FUNCTION_BLOCK FB_Bel
VAR_INPUT
	Freigabe_auto			: BOOL;
	Freigabe_Deakt_auto		: BOOL;
	Betrieb_Anford_auto		: BOOL;
	Steuerung_Sollw_auto	: REAL; (* 0-100*)
	Quittierung				: BOOL;
	Adresse					: BYTE;
	AdressType				: E_DALIV2AddrType;
END_VAR
VAR_OUTPUT
	Steuerung				: ST_Bel_Steuerung;
	Stellwert				: ST_Bel_Stellwert;
	Zustand					: ST_Bel_Zustand;
	Parameter				: ST_Bel_Parameter;
END_VAR
VAR
	Zustandscheck			: FB_Bel_Zustandscheck;
	Logik					: FB_Bel_Logik;
	Ablaufsteuerung			: FB_Bel_Ablaufsteuerung;
	Sollwertscheck			: FB_Bel_Sollwertscheck;
	SteuerungsVorgang		: FB_Bel_Steuerung;

	Stellwertscheck			: FB_Bel_Stellwertscheck;
	QuitTrig				: FB_SetResetFallTrigger;

	LeseDaten				: FB_Bel_Input;
	SchreibeDaten			: FB_Bel_Output;

	Dali_Dimmer				: FB_DALIV2Dimmer1Switch;
	Dali_Communication		: FB_DALIV2Communication;
	Dali_Off				: FB_DALIV2Off;
	Dali_ArcPower			: FB_DALIV2DirectArcPowerControl;

	OUT_Dali_Betrieb		: BOOL;
	OUT_Dali_Leistung		: BYTE;
	Dali_Error				: BOOL;
	Dali_Dimm_Betrieb		: BOOL:= FALSE;
	Dali_ErrorID			: UDINT;
	Dali_bBusy				: BOOL;
	Dali_bOn				: BOOL:=TRUE;
	Dali_bOff				: BOOL:=FALSE;
	Dali_TON				: TON;

	Dali_Arc_Busy			: BOOL;
	Dali_Arc_Error			: BOOL;
	Dali_Arc_ErrorID		: UDINT;

	Dali_Off_Busy			: BOOL;
	Dali_Off_Error			: BOOL;
	Dali_Off_ErrorID		: UDINT;

	IN_Leistung				: BYTE;
	IN_Dali_Arc_Error		: BOOL;
	IN_Dali_Off_Error		: BOOL;
	IN_Dali_Error			: BOOL;

	DALI_GetSettings		: FB_DALIV2GetSettings;
	DALI_Setting_Array		: ARRAY [0..63] OF ST_DALIV2DeviceSettings;
	Lampen_Monitoring		: FB_Bel_Monitoring;

END_VAR

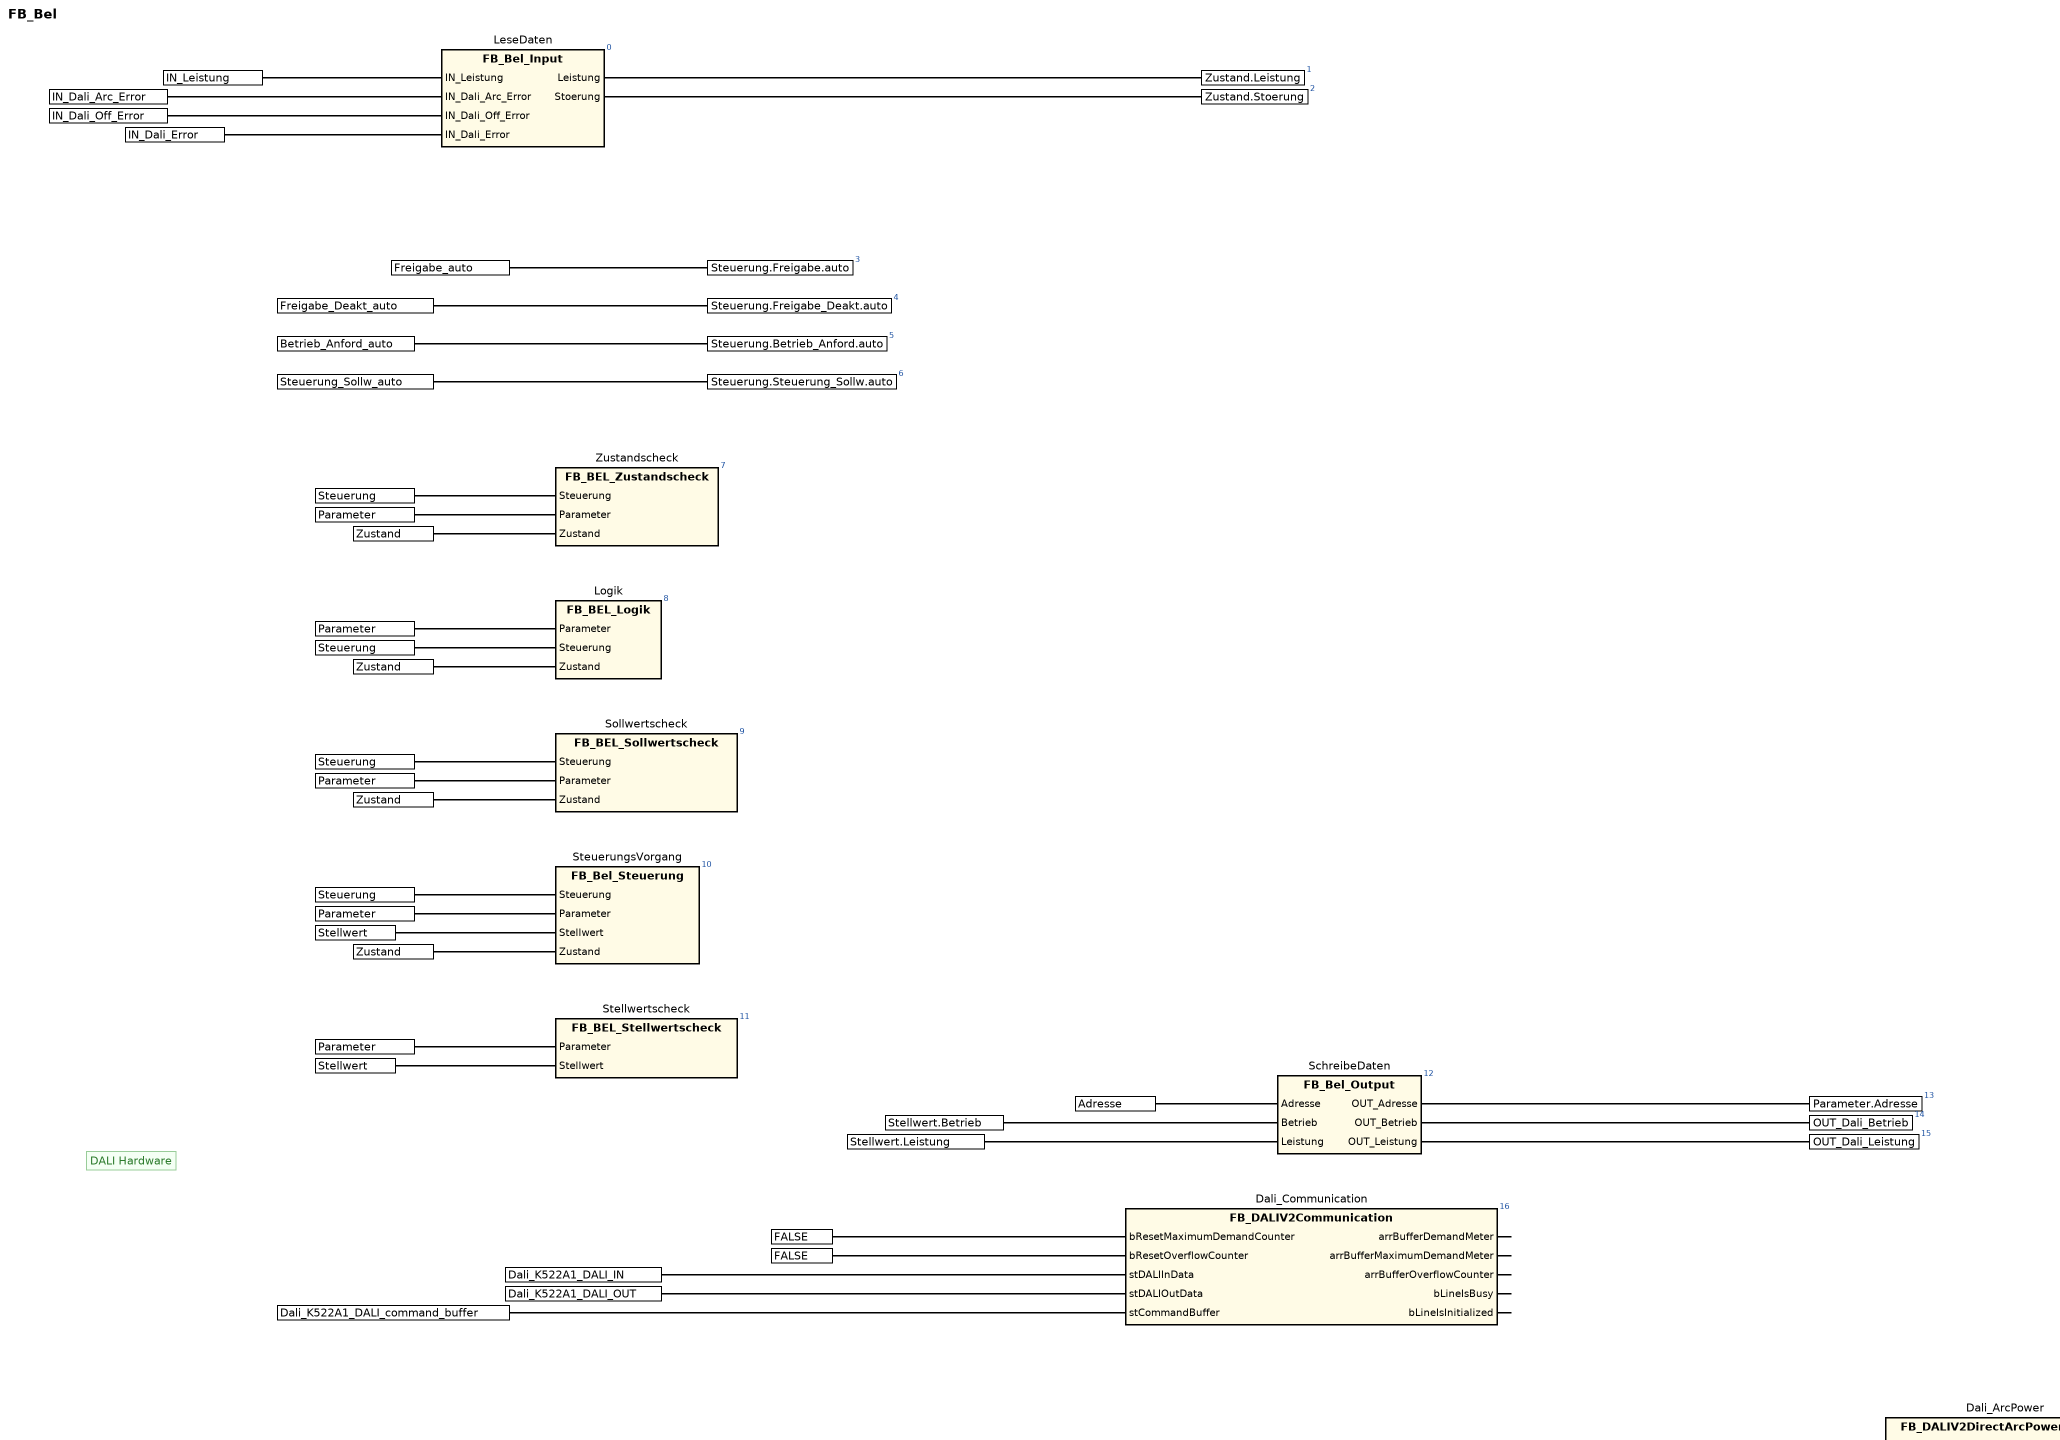
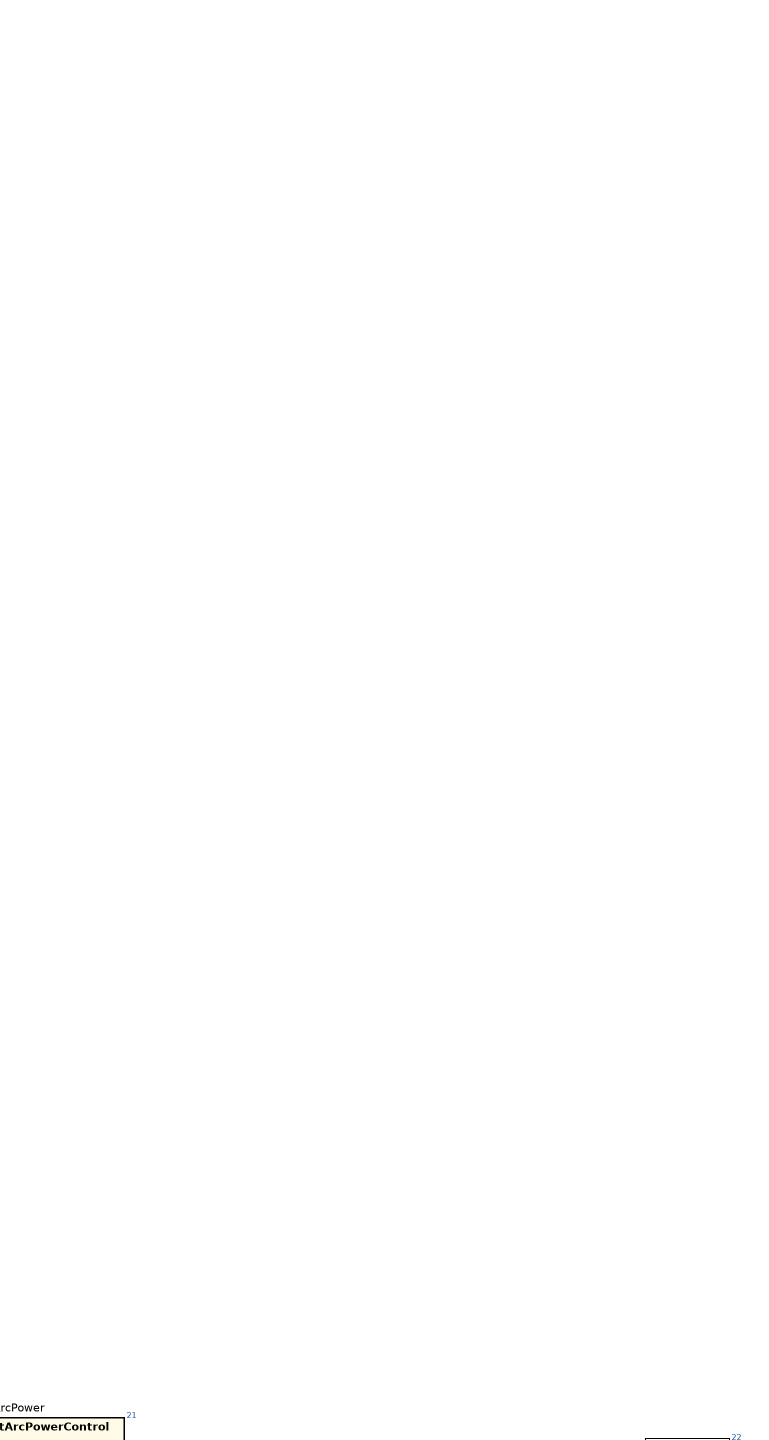
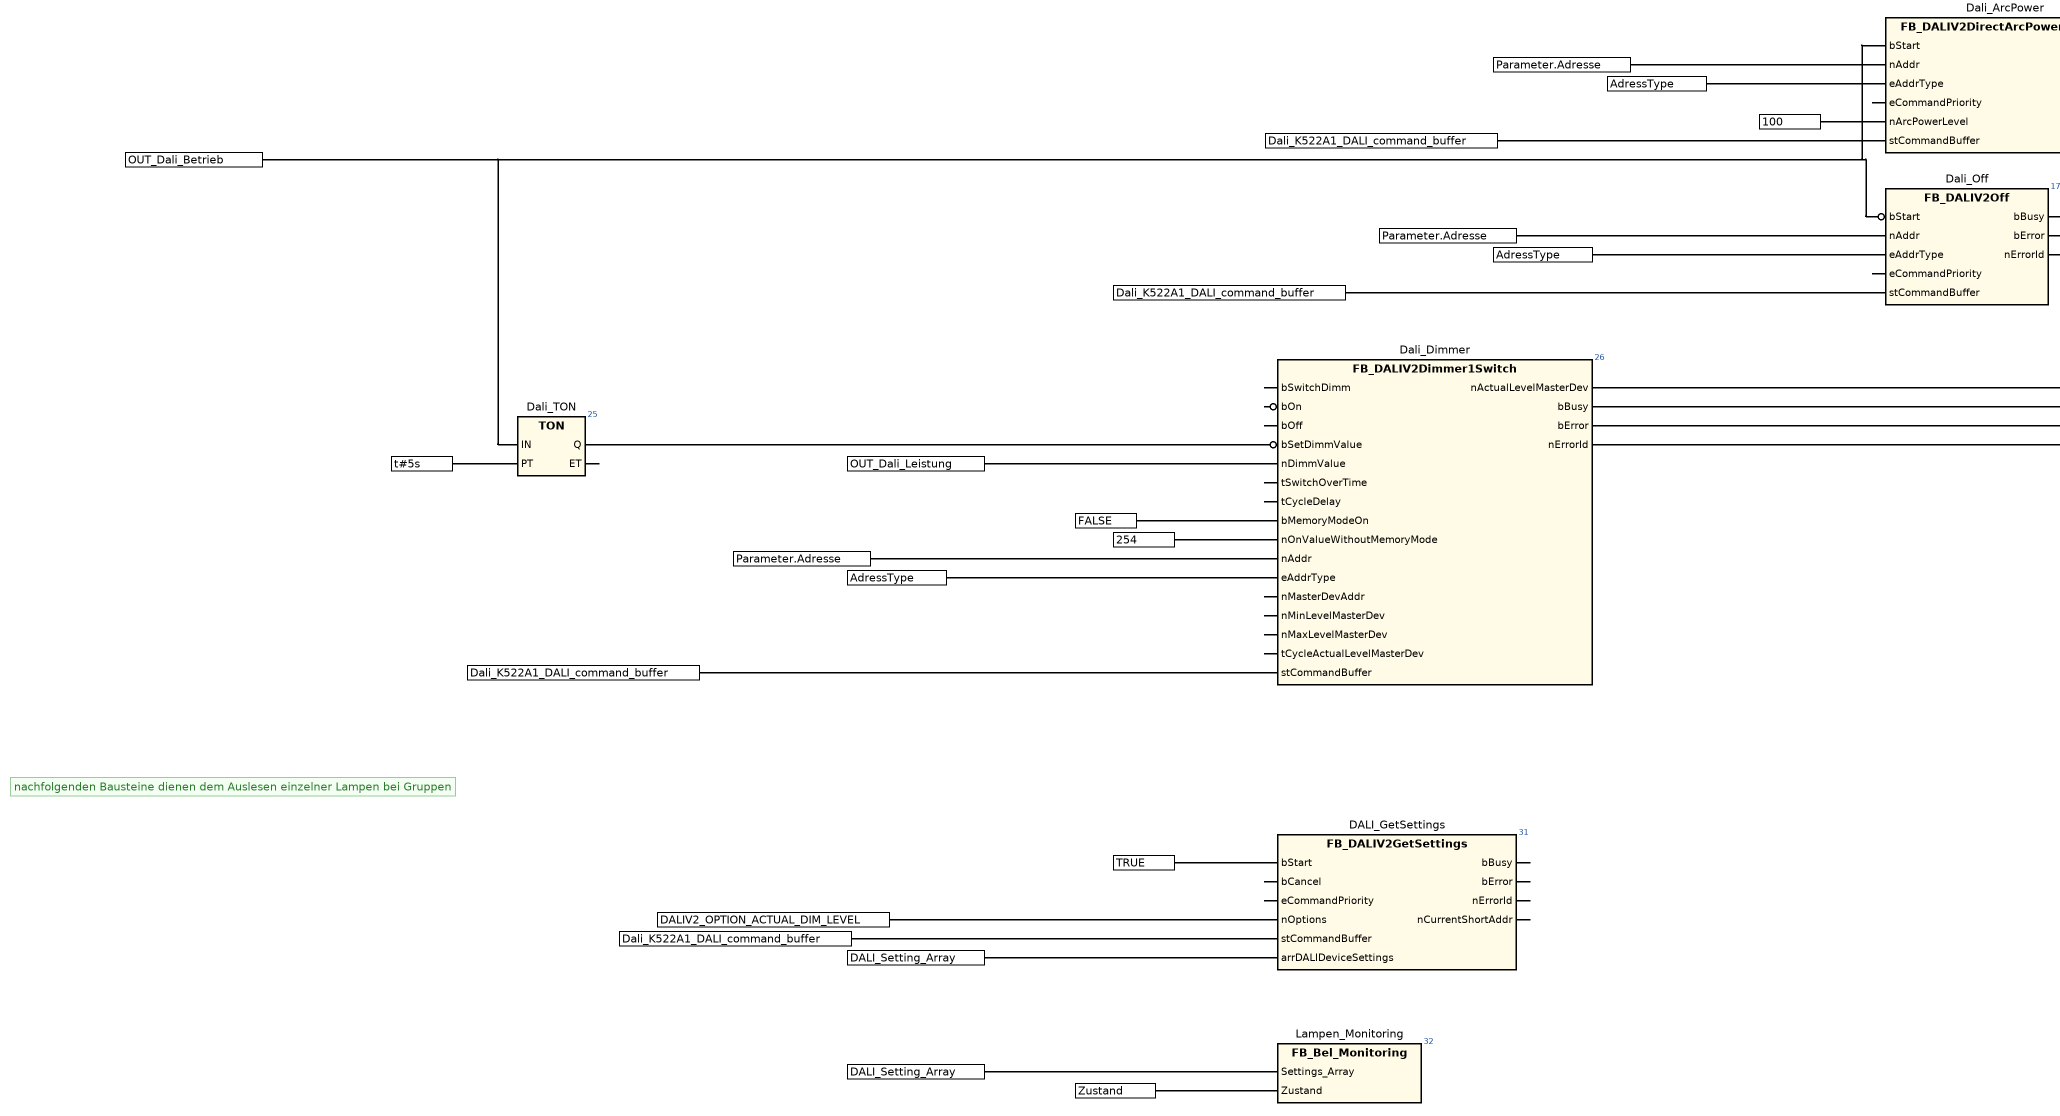
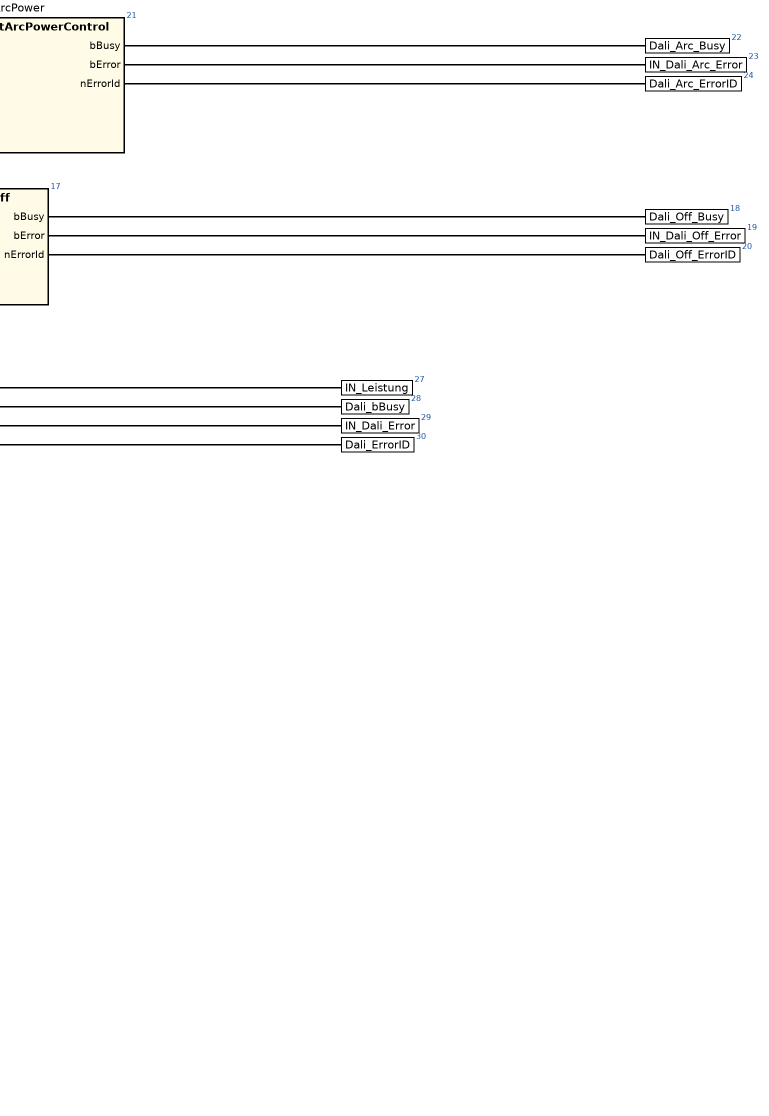
LeseDaten(
    IN_Leistung := IN_Leistung,
    IN_Dali_Arc_Error := IN_Dali_Arc_Error,
    IN_Dali_Off_Error := IN_Dali_Off_Error,
    IN_Dali_Error := IN_Dali_Error); // FB_Bel_Input
Zustand.Leistung := LeseDaten.Leistung;
Zustand.Stoerung := LeseDaten.Stoerung;
Steuerung.Freigabe.auto := Freigabe_auto;
Steuerung.Freigabe_Deakt.auto := Freigabe_Deakt_auto;
Steuerung.Betrieb_Anford.auto := Betrieb_Anford_auto;
Steuerung.Steuerung_Sollw.auto := Steuerung_Sollw_auto;
Zustandscheck(Steuerung := Steuerung, Parameter := Parameter, Zustand := Zustand); // FB_BEL_Zustandscheck
Logik(Parameter := Parameter, Steuerung := Steuerung, Zustand := Zustand); // FB_BEL_Logik
Sollwertscheck(Steuerung := Steuerung, Parameter := Parameter, Zustand := Zustand); // FB_BEL_Sollwertscheck
SteuerungsVorgang(Steuerung := Steuerung, Parameter := Parameter, Stellwert := Stellwert, Zustand := Zustand); // FB_Bel_Steuerung
Stellwertscheck(Parameter := Parameter, Stellwert := Stellwert); // FB_BEL_Stellwertscheck
SchreibeDaten(Adresse := Adresse, Betrieb := Stellwert.Betrieb, Leistung := Stellwert.Leistung); // FB_Bel_Output
Parameter.Adresse := SchreibeDaten.OUT_Adresse;
OUT_Dali_Betrieb := SchreibeDaten.OUT_Betrieb;
OUT_Dali_Leistung := SchreibeDaten.OUT_Leistung;
// DALI Hardware
Dali_Communication(
    bResetMaximumDemandCounter := FALSE,
    bResetOverflowCounter := FALSE,
    stDALIInData := Dali_K522A1_DALI_IN,
    stDALIOutData := Dali_K522A1_DALI_OUT,
    stCommandBuffer := Dali_K522A1_DALI_command_buffer); // FB_DALIV2Communication
Dali_Off(
    bStart := NOT OUT_Dali_Betrieb,
    nAddr := Parameter.Adresse,
    eAddrType := AdressType,
    stCommandBuffer := Dali_K522A1_DALI_command_buffer); // FB_DALIV2Off
Dali_Off_Busy := Dali_Off.bBusy;
IN_Dali_Off_Error := Dali_Off.bError;
Dali_Off_ErrorID := Dali_Off.nErrorId;
Dali_ArcPower(
    bStart := OUT_Dali_Betrieb,
    nAddr := Parameter.Adresse,
    eAddrType := AdressType,
    nArcPowerLevel := 100,
    stCommandBuffer := Dali_K522A1_DALI_command_buffer); // FB_DALIV2DirectArcPowerControl
Dali_Arc_Busy := Dali_ArcPower.bBusy;
IN_Dali_Arc_Error := Dali_ArcPower.bError;
Dali_Arc_ErrorID := Dali_ArcPower.nErrorId;
Dali_TON(IN := OUT_Dali_Betrieb, PT := t#5s); // TON
Dali_Dimmer(
    bSetDimmValue := NOT Dali_TON.Q,
    nDimmValue := OUT_Dali_Leistung,
    bMemoryModeOn := FALSE,
    nOnValueWithoutMemoryMode := 254,
    nAddr := Parameter.Adresse,
    eAddrType := AdressType,
    stCommandBuffer := Dali_K522A1_DALI_command_buffer); // FB_DALIV2Dimmer1Switch
IN_Leistung := Dali_Dimmer.nActualLevelMasterDev;
Dali_bBusy := Dali_Dimmer.bBusy;
IN_Dali_Error := Dali_Dimmer.bError;
Dali_ErrorID := Dali_Dimmer.nErrorId;
// nachfolgenden Bausteine dienen dem Auslesen einzelner Lampen bei Gruppen
DALI_GetSettings(
    bStart := TRUE,
    nOptions := DALIV2_OPTION_ACTUAL_DIM_LEVEL,
    stCommandBuffer := Dali_K522A1_DALI_command_buffer,
    arrDALIDeviceSettings := DALI_Setting_Array); // FB_DALIV2GetSettings
Lampen_Monitoring(Settings_Array := DALI_Setting_Array, Zustand := Zustand); // FB_Bel_Monitoring

END_FUNCTION_BLOCK

(* stored: Version 1.1.0.1, ProductVersion 3.1.4024.10
   POU FB_Bel: Id {cdb4ba03-987f-474a-95f9-59e5f292df0c}, SpecialFunc None *)
